// TIA Portal project "RADIO" (V11)

(* hardware
DEVICE "HMI_1"  KTP600 Basic PN
   slot 0: "HMI"  HMI  6AV6647-0AD11-3AX0  11.0.0
   slot 1: "HMI_RT_1"  KTP600 Basic PN  6AV6647-0AD11-3AX0  11.0.0
   slot 5: "IE_CP_1"  PROFINET interface  IE_CP  V7.1.0
      slot 1: "PROFINET_Interfaz_1"  HMI IE SUBMODULE
         slot 1: "PORT_1"  HMI IE PORTMODULE 1  1.0.0.0
DEVICE "S7300/ET200 station_1"  SIMATIC 300-Station
   slot 0: "Perfil soporte_0"  Rail  6ES7 390-1***0-0AA0
   slot 2: "PLC_1"  CPU 313C-2 DP  6ES7 313-6CF03-0AB0  V2.6
      slot 0: "Interfaz MPI_1"  MPI
      slot 1: "Interfaz DP_1"  DP
      slot 2: "DI16/DO16_1"  DI16/DO16
      slot 4: "Contaje_1"  Counter
   slot 4: "CP 343-1 Lean_1"  CP 343-1 LEAN  6GK7 343-1CX10-0XE0  V2.4
*)

// ===== PLC "PLC_1"  CPU 313C-2 DP =====

VAR_GLOBAL   // PLC tag table "Tabla de variables estándar"
   "DISPLAY M BIT 0" AT %M0.0 : Bool;
   "DISPLAY M BIT 1" AT %M0.1 : Bool;
   "DISPLAY M BIT 2" AT %M0.2 : Bool;
   "DISPLAY M BIT 3" AT %M0.3 : Bool;
   "DISPLAY M BIT 4" AT %M0.4 : Bool;
   "DISPLAY M BIT 5" AT %M0.5 : Bool;
   "DISPLAY M BIT 6" AT %M0.6 : Bool;
   "DISPLAY M SALIDA" AT %MB0 : Byte;
   "DISPLAY D BIT 0" AT %M1.0 : Bool;
   "DISPLAY D BIT 1" AT %M1.1 : Bool;
   "DISPLAY D BIT 2" AT %M1.2 : Bool;
   "DISPLAY D BIT 3" AT %M1.3 : Bool;
   "DISPLAY D BIT 4" AT %M1.4 : Bool;
   "DISPLAY D BIT 5" AT %M1.5 : Bool;
   "DISPLAY D BIT 6" AT %M1.6 : Bool;
   "DISPLAY D SALIDA" AT %MB1 : Byte;
   "DISPLAY U BIT 0" AT %M2.0 : Bool;
   "DISPLAY U BIT 1" AT %M2.1 : Bool;
   "DISPLAY U BIT 2" AT %M2.2 : Bool;
   "DISPLAY U BIT 3" AT %M2.3 : Bool;
   "DISPLAY U BIT 4" AT %M2.4 : Bool;
   "DISPLAY U BIT 5" AT %M2.5 : Bool;
   "DISPLAY U BIT 6" AT %M2.6 : Bool;
   "DISPLAY U SALIDA" AT %MB2 : Byte;
   "DISPLAY DE BIT 0" AT %M3.0 : Bool;
   "DISPLAY DE BIT 1" AT %M3.1 : Bool;
   "DISPLAY DE BIT 2" AT %M3.2 : Bool;
   "DISPLAY DE BIT 3" AT %M3.3 : Bool;
   "DISPLAY DE BIT 4" AT %M3.4 : Bool;
   "DISPLAY DE BIT 5" AT %M3.5 : Bool;
   "DISPLAY DE BIT 6" AT %M3.6 : Bool;
   "DISPLAY DE SALIDA" AT %MB3 : Byte;
   "DISPLAY CE BIT 0" AT %M4.0 : Bool;
   "DISPLAY CE BIT 1" AT %M4.1 : Bool;
   "DISPLAY CE BIT 2" AT %M4.2 : Bool;
   "DISPLAY CE BIT 3" AT %M4.3 : Bool;
   "DISPLAY CE BIT 4" AT %M4.4 : Bool;
   "DISPLAY CE BIT 5" AT %M4.5 : Bool;
   "DISPLAY CE BIT 6" AT %M4.6 : Bool;
   "DISPLAY CE SALIDA" AT %MB4 : Byte;
   "LED MEMORIA 1" AT %M5.0 : Bool;
   "LED MEMORIA 2" AT %M5.1 : Bool;
   "LED MEMORIA 3" AT %M5.2 : Bool;
   "LED MEMORIA 4" AT %M5.3 : Bool;
   "LED MEMORIA 5" AT %M5.4 : Bool;
   "LED MEMORIA 6" AT %M5.5 : Bool;
   "IZQUIERDA" AT %M5.6 : Bool;
   "DERECHA" AT %M6.7 : Bool;
   "MEMORIA 1" AT %M7.0 : Bool;
   "MEMORIA 2" AT %M7.1 : Bool;
   "MEMORIA 3" AT %M7.2 : Bool;
   "MEMORIA 4" AT %M7.3 : Bool;
   "MEMORIA 5" AT %M7.4 : Bool;
   "MEMORIA 6" AT %M7.5 : Bool;
   "ALMACENAJE M" AT %MD8 : DWord;
   "ALMACENAJE D" AT %MD12 : DWord;
   "ALMACENAJE U" AT %MD16 : DWord;
   "ALMACENAJE DE" AT %MD20 : DWord;
   "ALMACENAJE CE" AT %MD24 : DWord;
   "PARALELA M" AT %MD28 : DInt;
   "PARALELE D" AT %MD32 : DInt;
   "PARALELA DE" AT %MD36 : DInt;
   "PARALELA CE" AT %MD40 : DInt;
   "DISPLAY C BIT 1" AT %M44.0 : Bool;
   "DISPLAY C BIT 2" AT %M44.1 : Bool;
   "DISPALY C SALIDA" AT %MB44 : Byte;
   "INCREMENTO DE" AT %M45.0 : Bool;
   "DECREMERNTO DE" AT %M45.1 : Bool;
   "Tag_1" AT %A0.0 : Bool;
   "Tag_2" AT %A0.1 : Bool;
   "Tag_3" AT %E0.0 : Bool;
END_VAR

DATA_BLOCK "RADIO"   // DB1
{ S7_Optimized_Access := 'FALSE' }
VERSION : 0.1
   VAR
      PUNTERO : Array [0..10] of Byte;
      FLANCOS : Array [0..50] of Bool;
      BOBINAS : Array [0..50] of Bool;
      "NUMERO -1" : DInt := -1;
      "NUMERO -2" : DInt := -2;
   END_VAR
BEGIN
   PUNTERO[0] := B#16#3F;
   PUNTERO[1] := B#16#06;
   PUNTERO[2] := B#16#5B;
   PUNTERO[3] := B#16#4F;
   PUNTERO[4] := B#16#66;
   PUNTERO[5] := B#16#6D;
   PUNTERO[6] := B#16#7D;
   PUNTERO[7] := B#16#7;
   PUNTERO[8] := B#16#7F;
   PUNTERO[9] := B#16#6F;
END_DATA_BLOCK

FUNCTION "DISPLAY CE" : Void   // FC1, STL
TITLE = DISPLAY CE
{ S7_Optimized_Access := 'FALSE' }
VERSION : 0.1
// ESTE DISPLAY SOLO REPRESENTA LOS VALORES DE 0 Y 5 , SERA EL QUE GOBIERNE A LOS DEMAS CUANDO PASE DE 5 A 0 SUMARA UNA UNIDAD EN EL DISPLAY DE Y ASI SUCESIVAMANETE LA FRECUENCIA MINIMA SERA 87.00 Y LA MAXIMA 108.00.
   VAR_INPUT
      DERECHA : Bool;
      IZQUIERDA : Bool;
   END_VAR
   VAR_OUTPUT
      SALIDA : Byte;
      "INCREMENTO DE" : Bool;
      "DECREMENTO DE" : Bool;
   END_VAR
BEGIN

REGION Network 1: CREACION DEL PUNTERO
         AN    "RADIO".BOBINAS[0];
         FP    "RADIO".FLANCOS[0];
         JNB   _001;
         L     P#0.0;
         T     "ALMACENAJE CE";
   _001: NOP   0;
END_REGION

REGION Network 2: SUMA PARALELA DOBLE ENTERA..
   // LOS VALORES DEL PUNTERO VAN A SER 2 " 0 Y 5 " POR LO TANTO HAGO UNA SUMA PARALELA Y LUEGO PROGRAMO MEDIANTE COMPARADORES LAS CONDICIONES FINALMENTE TRANSFIERO EL RESULTADO AL PUNTERO.
         A     "DERECHA";
         FP    "RADIO".FLANCOS[1];
         JNB   _002;
         L     1;
         L     "PARALELA CE";
         +D;
         T     "PARALELA CE";
   _002: NOP   0;
END_REGION

REGION Network 3: RESTA PARALELA DOBLE ENTERA.
   // LOS VALORES DEL PUNTERO VAN A SER 2 " 0 Y 5 " POR LO TANTO HAGO UNA RESTA PARALELA Y LUEGO PROGRAMO MEDIANTE COMPARADORES LAS CONDICIONES FINALMENTE TRANSFIERO EL RESULTADO AL PUNTERO.
         A     "IZQUIERDA";
         FP    "RADIO".FLANCOS[2];
         JNB   _003;
         L     "PARALELA CE";
         L     1;
         -D;
         T     "PARALELA CE";
   _003: NOP   0;
END_REGION

REGION Network 4: RESET VARIABLE PARALELA CE.
   // CUANDO EL VALOR DE "PARALELLA CE " SEA =  2 TRANSFIERE UN 0 A LA MISMA VARIABLE.
         O(;
         L     2;
         L     "PARALELA CE";
         ==D;
         );
         O     "RADIO".BOBINAS[1];
         FP    "RADIO".FLANCOS[3];
         JNB   _004;
         L     0;
         T     "PARALELA CE";
   _004: NOP   0;
END_REGION

REGION Network 5: INCREMENTO DISPLAY DE.
   // ENVIA UN PULSO A LA SUMA DE EL DISPLAY DE PARA QUE INCREMENTE UNA UNDAD.
         A(;
         L     2;
         L     "PARALELA CE";
         ==D;
         );
         =     #"INCREMENTO DE";
END_REGION

REGION Network 6: CARGA DE LOS VALORES DEL LOS BYTES DEL DB1 EN UN BYTE DE SALIDA.
         AN    "RADIO".BOBINAS[0];
         JNB   _005;
         L     DBB [ "ALMACENAJE CE" ];
         T     #SALIDA;
   _005: NOP   0;
END_REGION

REGION Network 7: COMPARACION = 1.
   // CARGARA UN 5 Y EL PUNERO REPRESENTARA ESE NUMERO DEL DB1.
         O(;
         L     "PARALELA CE";
         L     1;
         ==D;
         );
         O     #"DECREMENTO DE";
         FP    "RADIO".FLANCOS[4];
         JNB   _006;
         L     P#5.0;
         T     "ALMACENAJE CE";
   _006: NOP   0;
END_REGION

REGION Network 8: COMPARACION = 0
   // CARGARA UN 0 Y EL PUNTERO REPRESENTARA ESE NUMERO DEL DB1.
         A(;
         L     "PARALELA CE";
         L     0;
         ==D;
         );
         FP    "RADIO".FLANCOS[5];
         JNB   _007;
         L     P#0.0;
         T     "ALMACENAJE CE";
   _007: NOP   0;
END_REGION

REGION Network 9: DECREMENTO DISPLAY DE EN NEGATIVO REPRESENTA 5
   // CUANDO EL VALOR DE LA VARIABLE MD40 SEA = -1 REPRESENTARA 5 EN DISPLAY CE
         A(;
         L     "PARALELA CE";
         L     "RADIO"."NUMERO -1";
         ==D;
         );
         FP    "RADIO".FLANCOS[8];
         =     #"DECREMENTO DE";
END_REGION

REGION Network 10: RESET CUANDO SEA = -2
   // PARA PODER SEGUIR CON EL DECREMRNTO Y ESTE SINCRONADO LA COMPARACION SERA = -2 ENVIANDO UN PULSO A LA FUNCION DE RESET
         A(;
         L     "PARALELA CE";
         L     "RADIO"."NUMERO -2";
         ==D;
         );
         =     "RADIO".BOBINAS[1];
END_REGION
END_FUNCTION

FUNCTION "DISPLAY DE" : Void   // FC2, STL
TITLE = DISPLAY DE.
{ S7_Optimized_Access := 'FALSE' }
VERSION : 0.1
// REPRESENTARA LOS NUMEROS DEL 0 AL 9 ,
   VAR_INPUT
      "INCREMENTO DE" : Bool;
      "DECREMENTO DE" : Bool;
   END_VAR
   VAR_OUTPUT
      SALIDA : Byte;
   END_VAR
BEGIN

REGION Network 1: CREACION DEL PUNTERO.
         AN    "RADIO".BOBINAS[0];
         FP    "RADIO".FLANCOS[6];
         JNB   _001;
         L     P#0.0;
         T     "ALMACENAJE DE";
   _001: NOP   0;
END_REGION

REGION Network 2: INCREMENTO DEL PUNTERO
   // INCREMENTARA MEDIANTE LOS PULSOS QUE ENVIA EL DISPALY CE CUANDO = 2.
         A     #"INCREMENTO DE";
         FP    "RADIO".FLANCOS[7];
         JNB   _002;
         L     P#1.0;
         L     "ALMACENAJE DE";
         +D;
         T     "ALMACENAJE DE";
   _002: NOP   0;
END_REGION

REGION Network 5: CARGA DE LOS VALORES DEL LOS BYTES DEL DB1 EN UN BYTE DE SALIDA.
         AN    "RADIO".BOBINAS[0];
         JNB   _003;
         L     DBB [ "ALMACENAJE DE"];
         T     #SALIDA;
   _003: NOP   0;
END_REGION
END_FUNCTION

ORGANIZATION_BLOCK "Main"   // OB1, STL
TITLE = "Main Program Sweep (Cycle)"
{ S7_Optimized_Access := 'FALSE' }
VERSION : 0.1
   VAR_TEMP
      OB1_EV_CLASS : Byte;   // Bits 0-3 = 1 (Coming event), Bits 4-7 = 1 (Event class 1)
      OB1_SCAN_1 : Byte;   // 1 (Cold restart scan 1 of OB 1), 3 (Scan 2-n of OB 1)
      OB1_PRIORITY : Byte;   // Priority of OB Execution
      OB1_OB_NUMBR : Byte;   // 1 (Organization block 1, OB1)
      OB1_RESERVED_1 : Byte;   // Reserved for system
      OB1_RESERVED_2 : Byte;   // Reserved for system
      OB1_PREV_CYCLE : Int;   // Cycle time of previous OB1 scan (milliseconds)
      OB1_MIN_CYCLE : Int;   // Minimum cycle time of OB1 (milliseconds)
      OB1_MAX_CYCLE : Int;   // Maximum cycle time of OB1 (milliseconds)
      OB1_DATE_TIME : Date_And_Time;   // Date and time OB1 started
   END_VAR
BEGIN

REGION Network 1: APERTURA DEL DB1.
         OPN   "RADIO";
END_REGION

REGION Network 2: LLAMADA FC1. DISPLAY CE.
         CALL  "DISPLAY CE"
         ( DERECHA         := "IZQUIERDA",
           IZQUIERDA       := "DERECHA",
           SALIDA          := "DISPLAY CE SALIDA",
           "INCREMENTO DE" := "INCREMENTO DE",
           "DECREMENTO DE" := "DECREMERNTO DE"
         );
END_REGION

REGION Network 3: LLAMDA FC2. DISPLAY DE
         CALL  "DISPLAY DE"
         ( "INCREMENTO DE" := "INCREMENTO DE",
           "DECREMENTO DE" := "DECREMERNTO DE",
           SALIDA          := "DISPLAY DE SALIDA"
         );
END_REGION

REGION Network 4
         A     "INCREMENTO DE";
         S     "Tag_1";
END_REGION
END_ORGANIZATION_BLOCK

(* ===== HMI "HMI_RT_1" =====
connection "Conexión_HMI": ETHERNET, SIMATIC S7 300/400 MPI

HMI tags "Tabla de variables estándar"
   "DISPLAY M BIT 1" : Bool = PLC "DISPLAY M BIT 1", 1 s
   "DISPLAY M BIT 2" : Bool = PLC "DISPLAY M BIT 2", 1 s
   "DISPLAY M BIT 3" : Bool = PLC "DISPLAY M BIT 3", 1 s
   "DISPLAY M BIT 4" : Bool = PLC "DISPLAY M BIT 4", 1 s
   "DISPLAY M BIT 5" : Bool = PLC "DISPLAY M BIT 5", 1 s
   "DISPLAY M BIT 6" : Bool = PLC "DISPLAY M BIT 6", 1 s
   "DISPLAY M BIT 0" : Bool = PLC "DISPLAY M BIT 0", 1 s
   "DISPLAY U BIT 0" : Bool = PLC "DISPLAY U BIT 0", 1 s
   "DISPLAY U BIT 1" : Bool = PLC "DISPLAY U BIT 1", 1 s
   "DISPLAY U BIT 2" : Bool = PLC "DISPLAY U BIT 2", 1 s
   "DISPLAY U BIT 3" : Bool = PLC "DISPLAY U BIT 3", 1 s
   "DISPLAY U BIT 4" : Bool = PLC "DISPLAY U BIT 4", 1 s
   "DISPLAY U BIT 5" : Bool = PLC "DISPLAY U BIT 5", 1 s
   "DISPLAY U BIT 6" : Bool = PLC "DISPLAY U BIT 6", 1 s
   "IZQUIERDA" : Bool = PLC "IZQUIERDA", 1 s
   "LED MEMORIA 1" : Bool = PLC "LED MEMORIA 1", 1 s
   "DISPLAY D BIT 0" : Bool = PLC "DISPLAY D BIT 0", 1 s
   "DISPLAY D BIT 2" : Bool = PLC "DISPLAY D BIT 2", 1 s
   "DISPLAY D BIT 1" : Bool = PLC "DISPLAY D BIT 1", 1 s
   "DISPLAY D BIT 3" : Bool = PLC "DISPLAY D BIT 3", 1 s
   "DISPLAY D BIT 4" : Bool = PLC "DISPLAY D BIT 4", 1 s
   "DISPLAY D BIT 5" : Bool = PLC "DISPLAY D BIT 5", 1 s
   "DISPLAY D BIT 6" : Bool = PLC "DISPLAY D BIT 6", 1 s
   "DISPLAY DE BIT 0" : Bool = PLC "DISPLAY DE BIT 0", 1 s
   "DISPLAY DE BIT 1" : Bool = PLC "DISPLAY DE BIT 1", 1 s
   "DISPLAY DE BIT 2" : Bool = PLC "DISPLAY DE BIT 2", 1 s
   "DISPLAY DE BIT 3" : Bool = PLC "DISPLAY DE BIT 3", 1 s
   "DISPLAY DE BIT 4" : Bool = PLC "DISPLAY DE BIT 4", 1 s
   "DISPLAY DE BIT 5" : Bool = PLC "DISPLAY DE BIT 5", 1 s
   "DISPLAY DE BIT 6" : Bool = PLC "DISPLAY DE BIT 6", 1 s
   "DISPLAY CE BIT 0" : Bool = PLC "DISPLAY CE BIT 0", 1 s
   "DISPLAY CE BIT 1" : Bool = PLC "DISPLAY CE BIT 1", 1 s
   "DISPLAY CE BIT 2" : Bool = PLC "DISPLAY CE BIT 2", 1 s
   "DISPLAY CE BIT 3" : Bool = PLC "DISPLAY CE BIT 3", 1 s
   "DISPLAY CE BIT 4" : Bool = PLC "DISPLAY CE BIT 4", 1 s
   "DISPLAY CE BIT 5" : Bool = PLC "DISPLAY CE BIT 5", 1 s
   "DISPLAY CE BIT 6" : Bool = PLC "DISPLAY CE BIT 6", 1 s
   "LED MEMORIA 2" : Bool = PLC "LED MEMORIA 2", 1 s
   "LED MEMORIA 3" : Bool = PLC "LED MEMORIA 3", 1 s
   "LED MEMORIA 4" : Bool = PLC "LED MEMORIA 4", 1 s
   "LED MEMORIA 5" : Bool = PLC "LED MEMORIA 5", 1 s
   "LED MEMORIA 6" : Bool = PLC "LED MEMORIA 6", 1 s
   "DERECHA" : Bool = PLC "DERECHA", 1 s
   "MEMORIA 1" : Bool = PLC "MEMORIA 1", 1 s
   "MEMORIA 2" : Bool = PLC "MEMORIA 2", 1 s
   "MEMORIA 3" : Bool = PLC "MEMORIA 3", 1 s
   "MEMORIA 4" : Bool = PLC "MEMORIA 4", 1 s
   "MEMORIA 5" : Bool = PLC "MEMORIA 5", 1 s
   "MEMORIA 6" : Bool = PLC "MEMORIA 6", 1 s
   "DISPLAY C BIT 1" : Bool = PLC "DISPLAY C BIT 1", 1 s
   "DISPLAY C BIT 2" : Bool = PLC "DISPLAY C BIT 2", 1 s

screen "Imagen_1" 320x240
   Button "Botón_1" at 7,195 size 45x40
   Button "Botón_2" at 56,195 size 45x40
   Button "Botón_3" at 110,195 size 25x25
   Button "Botón_4" at 143,195 size 25x25
   Button "Botón_5" at 176,195 size 25x25
   Button "Botón_6" at 209,195 size 25x25
   Button "Botón_7" at 241,195 size 25x25
   Button "Botón_8" at 272,195 size 25x25
*)